{attribute 'global_init_slot' := '40510'}
VAR_GLOBAL
  LblAgg_FunctionallyIndependentEequipment                 :FB_BA_Label:=( sObjName:='FEE', sDescr:='Funktional eigenständige Einrichtung');
  LblAgg_SelfContainedControlUnit                          :FB_BA_Label:=( sObjName:='ASR', sDescr:='Autarke Steuer- oder Regeleinheit');
  LblAgg_ControlCabinet                                    :FB_BA_Label:=( sObjName:='SSK', sDescr:='Schaltschrank (gewerkespezifisch)');
//     330 Türen, Tore, Fenster, Sonnenschutz
  LblAgg_WindowDrive                                       :FB_BA_Label:=( sObjName:='FEN', sDescr:='Fenster (Antrieb)');
  LblAgg_WindowContact                                     :FB_BA_Label:=( sObjName:='FEK', sDescr:='Fensterkontakt');
  LblAgg_Blind                                             :FB_BA_Label:=( sObjName:='JAL', sDescr:='Jalousie');
  LblAgg_Awning                                            :FB_BA_Label:=( sObjName:='MAR', sDescr:='Markise');
  LblAgg_RollerShutters                                    :FB_BA_Label:=( sObjName:='ROL', sDescr:='Rollläden');
  LblAgg_Gate                                              :FB_BA_Label:=( sObjName:='TOR', sDescr:='Tor');
  LblAgg_Door                                              :FB_BA_Label:=( sObjName:='TÜR', sDescr:='Tür');
  LblAgg_DoorContact                                       :FB_BA_Label:=( sObjName:='TÜK', sDescr:='Türkontakt');
  LblAgg_Blackout                                          :FB_BA_Label:=( sObjName:='VER', sDescr:='Verdunklung');
//     412 Wasseranlagen
  LblAgg_TraceHeating                                      :FB_BA_Label:=( sObjName:='BGH', sDescr:='Begleitheizung');
  LblAgg_ElectricHeating                                   :FB_BA_Label:=( sObjName:='EWH', sDescr:='Elektroheizung (TWW–Bereitung)');
  LblAgg_WaterFilter                                       :FB_BA_Label:=( sObjName:='WFL', sDescr:='Wasserfilter');
//     421 Wärmeerzeugungsanlagen
  LblAgg_Furnace                                           :FB_BA_Label:=( sObjName:='HZK', sDescr:='Heizkessel');
  LblAgg_HeatExchanger                                     :FB_BA_Label:=( sObjName:='WÜT', sDescr:='Wärmeübertrager');
//     430 Lufttechnische Anlagen und Kälteanlagen
  LblAgg_FanExhaustAir                                     :FB_BA_Label:=( sObjName:='FOV', sDescr:='Fortluftventilator');
  LblAgg_Airwasher                                         :FB_BA_Label:=( sObjName:='LWS', sDescr:='Luftwäscher');
  LblAgg_Humidifier                                        :FB_BA_Label:=( sObjName:='BEF', sDescr:='Befeuchter');
  LblAgg_HumidifierPump                                    :FB_BA_Label:=( sObjName:='BFP', sDescr:='Befeuchterpumpe');
  LblAgg_FireDamper                                        :FB_BA_Label:=( sObjName:='BSK', sDescr:='Brandschutzklappe, -ventil');
  LblAgg_SmokeProtectionDamper                             :FB_BA_Label:=( sObjName:='RSK', sDescr:='Rauchschutzklappe');
  LblAgg_SmokeExtractorDamper                              :FB_BA_Label:=( sObjName:='ERK', sDescr:='Entrauchungsklappe');
  LblAgg_CeilingSwirlDiffuser                              :FB_BA_Label:=( sObjName:='DDA', sDescr:='Deckendrallauslass');
  LblAgg_RoofAirHeater                                     :FB_BA_Label:=( sObjName:='DLA', sDescr:='Deckenlufterhitzer');
  LblAgg_DirectEvaporator                                  :FB_BA_Label:=( sObjName:='DVD', sDescr:='Direktverdampfer');
  LblAgg_ElectricalAirHeater                               :FB_BA_Label:=( sObjName:='ELH', sDescr:='Elektrolufterhitzer');
  LblAgg_ElectricReHeater                                  :FB_BA_Label:=( sObjName:='ENH', sDescr:='Elektronacherhitzer');
  LblAgg_ElectricaPreHeater                                :FB_BA_Label:=( sObjName:='EVH', sDescr:='Elektrovorerhitzer');
  LblAgg_HeaterGeneral                                     :FB_BA_Label:=( sObjName:='ERH', sDescr:='Erhitzer');
  LblAgg_FanExtractAir                                     :FB_BA_Label:=( sObjName:='ABV', sDescr:='Abluftventilator');
  LblAgg_InductionDevice                                   :FB_BA_Label:=( sObjName:='IND', sDescr:='Induktionsgerät');
  LblAgg_RefrigerantDryer                                  :FB_BA_Label:=( sObjName:='KTR', sDescr:='Kältetrockner');
  LblAgg_CirculatorySystem                                 :FB_BA_Label:=( sObjName:='KVS', sDescr:='KVS (WRG über Kreislaufverbundsysteme)');
  LblAgg_AirFilterOutsideAir                               :FB_BA_Label:=( sObjName:='LFI', sDescr:='Außenluftfilter');
  LblAgg_AirFilterSupplyAir                                :FB_BA_Label:=( sObjName:='LFI', sDescr:='Zuluftfilter');
  LblAgg_AirFilterExhaustAir                               :FB_BA_Label:=( sObjName:='LFI', sDescr:='Fortluftfilter');
  LblAgg_AirFilterExtractAir                               :FB_BA_Label:=( sObjName:='LFI', sDescr:='Abluftfilter');
  LblAgg_AirFilter                                         :FB_BA_Label:=( sObjName:='LFI', sDescr:='Luftfilter');
  LblAgg_VentilationDamper                                 :FB_BA_Label:=( sObjName:='LKL', sDescr:='Lüftungsklappe');
  LblAgg_VentilationDamperOutsideAir                       :FB_BA_Label:=( sObjName:='LKL', sDescr:='Außenluftklappe');
  LblAgg_VentilationDamperExhaustAir                       :FB_BA_Label:=( sObjName:='LKL', sDescr:='Fortluftklappe');
  LblAgg_VentilationDamperMixAir                           :FB_BA_Label:=( sObjName:='LKL', sDescr:='Mischluftklappe');
  LblAgg_VentilationDamperSupplyAir                        :FB_BA_Label:=( sObjName:='LKL', sDescr:='Zuluftklappe');
  LblAgg_VentilationDamperBypassAir                        :FB_BA_Label:=( sObjName:='LKL', sDescr:='Bypassklappe');
  LblAgg_Pump                                              :FB_BA_Label:=( sObjName:='PPE', sDescr:='Pumpe');
  LblAgg_RecirculatingAirCoolingDevice                     :FB_BA_Label:=( sObjName:='ULK', sDescr:='Umluftkühlgerät');
  LblAgg_FanRecirculatingAir                               :FB_BA_Label:=( sObjName:='UMV', sDescr:='Umluftventilator');
  LblAgg_UvFilter                                          :FB_BA_Label:=( sObjName:='UVF', sDescr:='UV-Filter');
  LblAgg_VariableFlowRateController                        :FB_BA_Label:=( sObjName:='VVR', sDescr:='Variabler Volumenstromregler');
  LblAgg_WaterAirHeater                                    :FB_BA_Label:=( sObjName:='WLH', sDescr:='Wasserlufterhitzer');
  LblAgg_WaterReHeater                                     :FB_BA_Label:=( sObjName:='WNH', sDescr:='Wassernacherhitzer');
  LblAgg_WaterPreHeater                                    :FB_BA_Label:=( sObjName:='WVH', sDescr:='Wasservorerhitzer');
  LblAgg_HeatRecovery                                      :FB_BA_Label:=( sObjName:='WRG', sDescr:='Wärmerückgewinnung');
  LblAgg_FanSupplyAir                                      :FB_BA_Label:=( sObjName:='ZUV', sDescr:='Zuluftventilator');
  LblAgg_SmokeExtractionSystems                            :FB_BA_Label:=( sObjName:='ERA', sDescr:='Entrauchungsanlagen');
  LblAgg_SmokeExtractionVentilator                         :FB_BA_Label:=( sObjName:='ERV', sDescr:='Entrauchungsventilator');
  LblAgg_VentWindow                                        :FB_BA_Label:=( sObjName:='NSF', sDescr:='Nachströmfenster');
  LblAgg_VentFlap                                          :FB_BA_Label:=( sObjName:='NSK', sDescr:='Nachströmklappe');
  LblAgg_VentDoor                                          :FB_BA_Label:=( sObjName:='NST', sDescr:='Nachströmtür');
  LblAgg_WakeFan                                           :FB_BA_Label:=( sObjName:='NSV', sDescr:='Nachströmventilator');
//     434 Kälteanlagen
  LblAgg_GlycoOilProtector                                 :FB_BA_Label:=( sObjName:='GLP', sDescr:='Glykol/Ölprotektor');
  LblAgg_Chiller                                           :FB_BA_Label:=( sObjName:='KMA', sDescr:='Kältemaschine');
  LblAgg_ReCoolingPlant                                    :FB_BA_Label:=( sObjName:='RKW', sDescr:='Rückkühlwerk');
//     440 Starkstromanlagen
  LblAgg_GeneralPowerSupply                                :FB_BA_Label:=( sObjName:='ASV', sDescr:='Allgemeine Spannungsversorgung');
  LblAgg_CombindeHeatPowerStation                          :FB_BA_Label:=( sObjName:='BHK', sDescr:='Blockheizkraftwerk');
  LblAgg_CompensationSystem                                :FB_BA_Label:=( sObjName:='KOA', sDescr:='Kompensationsanlage');
  LblAgg_CouplingSwitch                                    :FB_BA_Label:=( sObjName:='KUS', sDescr:='Kuppelschalter');
  LblAgg_LoadBreakSwitch                                   :FB_BA_Label:=( sObjName:='LTS', sDescr:='Lasttrennschalter');
  LblAgg_CircuitBreaker                                    :FB_BA_Label:=( sObjName:='LSS', sDescr:='Leistungsschalter');
  LblAgg_NetworkAnalyser                                   :FB_BA_Label:=( sObjName:='NAG', sDescr:='Netzanalysegerät');
  LblAgg_EmergencyPoweGeneratorUnit                        :FB_BA_Label:=( sObjName:='NSG', sDescr:='Notstromaggregat');
  LblAgg_EmergencyLighting                                 :FB_BA_Label:=( sObjName:='SIB', sDescr:='Sicherheitsbeleuchtung');
  LblAgg_SafetyPowerSupply                                 :FB_BA_Label:=( sObjName:='SSV', sDescr:='Sicherheitsspannungsversorgung');
  LblAgg_Transformer                                       :FB_BA_Label:=( sObjName:='TRF', sDescr:='Transformator');
  LblAgg_UninterruptiblePowerSupply                        :FB_BA_Label:=( sObjName:='USV', sDescr:='Unterbrechungsfreie Spannungsversorgung');
//     450 Fernmelde- und informationstechnische Anlagen
  LblAgg_CentralFireAlarmSystem                            :FB_BA_Label:=( sObjName:='BMZ', sDescr:='Brandmeldezentrale');
  LblAgg_FireControlPanel                                  :FB_BA_Label:=( sObjName:='FWT', sDescr:='Feuerwehrtableau');
  LblAgg_KitchenTableau                                    :FB_BA_Label:=( sObjName:='KÜT', sDescr:='Küchentableau');
  LblAgg_SmokeDetector                                     :FB_BA_Label:=( sObjName:='RME', sDescr:='Rauchmelder');
  LblAgg_SmokeProtectionScreen                             :FB_BA_Label:=( sObjName:='RSV', sDescr:='Rauchschutzvorhang');
  LblAgg_VoiceAlarmCentre                                  :FB_BA_Label:=( sObjName:='SAZ', sDescr:='Sprachalarmierungszentrale');
  LblAgg_Tableau                                           :FB_BA_Label:=( sObjName:='TBL', sDescr:='Tableau (allgemein)');
//     460 Förderanlagen
  LblAgg_LiftGeneral                                       :FB_BA_Label:=( sObjName:='AZA', sDescr:='Aufzug allgemein');
  LblAgg_GoodsLift                                         :FB_BA_Label:=( sObjName:='AZL', sDescr:='Lastenaufzug');
  LblAgg_PassengerLift                                     :FB_BA_Label:=( sObjName:='AZP', sDescr:='Personenaufzug');
//     470 Nutzerspezifische Anlagen
  LblAgg_FumeCupboard                                      :FB_BA_Label:=( sObjName:='DIG', sDescr:='Digestorium');
  LblAgg_Compressor                                        :FB_BA_Label:=( sObjName:='KOM', sDescr:='Kompressor');
  LblAgg_ProgrammableLogicControllers                      :FB_BA_Label:=( sObjName:='SPS', sDescr:='Speicherprogrammierbare Steuerung');
//     479 Nutzerspezifische Anlage, Wetterstation
  LblAgg_RainSensor                                        :FB_BA_Label:=( sObjName:='RGM', sDescr:='Regenmelder');
  LblAgg_SolarRadiation                                    :FB_BA_Label:=( sObjName:='SES', sDescr:='Sonneneinstrahlung');
  LblAgg_WeatherStation                                    :FB_BA_Label:=( sObjName:='WST', sDescr:='Wetterstation');
  LblAgg_WindSpeed                                         :FB_BA_Label:=( sObjName:='WDG', sDescr:='Windgeschwindigkeit');
  LblAgg_WindDirection                                     :FB_BA_Label:=( sObjName:='WDR', sDescr:='Windrichtung');
  LblAgg_WindForce                                         :FB_BA_Label:=( sObjName:='WDS', sDescr:='Windstärke');
  LblAgg_Brightness                                        :FB_BA_Label:=( sObjName:='HEL', sDescr:='Helligkeit');
  LblAgg_Dawn                                              :FB_BA_Label:=( sObjName:='HED', sDescr:='Dämmerungshelligkeit');
  LblAgg_PressureAbsolute                                  :FB_BA_Label:=( sObjName:='LUA', sDescr:='Luftdruck absolut');
  LblAgg_PressureRelative                                  :FB_BA_Label:=( sObjName:='LUR', sDescr:='Luftdruck relativ');
  LblAgg_GeoLatitude                                       :FB_BA_Label:=( sObjName:='BRG', sDescr:='Breitengrad');
  LblAgg_GeoLongitude                                      :FB_BA_Label:=( sObjName:='LAG', sDescr:='Längengrad');
  LblAgg_SunAzimuth                                        :FB_BA_Label:=( sObjName:='SST', sDescr:='Sonnenstand');
  LblAgg_SunElevation                                      :FB_BA_Label:=( sObjName:='SEL', sDescr:='Elevation');
  LblAgg_WeatherStationReset                               :FB_BA_Label:=( sObjName:='ALS', sDescr:='Wetterstation Reset');
  LblAgg_WeatherStationCommReset                           :FB_BA_Label:=( sObjName:='ALS', sDescr:='Wetterstation Reset serielle Kommunikation');
  LblAgg_WeatherStationComm                                :FB_BA_Label:=( sObjName:='WST', sDescr:='Wetterstation Kommunikation');
//     480 Gebäudeautomation
  LblAgg_SystemSwitch                                      :FB_BA_Label:=( sObjName:='ANL', sDescr:='Anlagenschalter');
  LblAgg_AutomationStationEquipment                        :FB_BA_Label:=( sObjName:='ASE', sDescr:='Automationsstationseinrichtung');
  LblAgg_BusLineCoupler                                    :FB_BA_Label:=( sObjName:='BUS', sDescr:='Bus-Linien-Koppler');
  LblAgg_DataInterfaceUnit                                 :FB_BA_Label:=( sObjName:='DSE', sDescr:='Datenschnittstelleneinheit');
  LblAgg_FieldbusModule                                    :FB_BA_Label:=( sObjName:='FBM', sDescr:='Feldbusmodul');
  LblAgg_InformationFocalPoint                             :FB_BA_Label:=( sObjName:='ISP', sDescr:='Informationsschwerpunkt');
  LblAgg_ManagementAndControlEquipment                     :FB_BA_Label:=( sObjName:='MBE', sDescr:='Management- und Bedieneinrichtung');
//     481 GA-Sensorik – Temperatur
  LblAgg_TemperatureGasEmission                            :FB_BA_Label:=( sObjName:='TAG', sDescr:='Abgastemperatur');
  LblAgg_TemperatureExtractAir                             :FB_BA_Label:=( sObjName:='TAB', sDescr:='Ablufttemperatur');
  LblAgg_TemperatureOutside                                :FB_BA_Label:=( sObjName:='TAU', sDescr:='Außentemperatur');
  LblAgg_TemperatureExhaustAir                             :FB_BA_Label:=( sObjName:='TFO', sDescr:='Fortlufttemperatur');
  LblAgg_FrostProtectionMonitor                            :FB_BA_Label:=( sObjName:='FSW', sDescr:='Frostschutzwächter');
  LblAgg_TemperatureMixedAir                               :FB_BA_Label:=( sObjName:='TMI', sDescr:='Mischlufttemperatur');
  LblAgg_TemperatureRoomAir                                :FB_BA_Label:=( sObjName:='TRU', sDescr:='Raumtemperatur');
  LblAgg_TemperatureReturnFlow                             :FB_BA_Label:=( sObjName:='TRL', sDescr:='Rücklauftemperatur');
  LblAgg_LimiterSafetyTemperature                          :FB_BA_Label:=( sObjName:='STB', sDescr:='Sicherheitstemperaturbegrenzer');
  LblAgg_MonitorSafetyTemperature                          :FB_BA_Label:=( sObjName:='STW', sDescr:='Sicherheitstemperaturwächter');
  LblAgg_TemperatureStorage                                :FB_BA_Label:=( sObjName:='TSP', sDescr:='Speichertemperatur');
  LblAgg_TemperatureDewPoint                               :FB_BA_Label:=( sObjName:='TTP', sDescr:='Taupunkttemperatur');
  LblAgg_MonitorDewPoint                                   :FB_BA_Label:=( sObjName:='TPW', sDescr:='Taupunktwächter');
  LblAgg_TemperatureAfterCooler                            :FB_BA_Label:=( sObjName:='TNK', sDescr:='Temperatur nach Kühler');
  LblAgg_TemperatureAfterPreHeater                         :FB_BA_Label:=( sObjName:='TNV', sDescr:='Temperatur nach Vorerhitzer');
  LblAgg_TemperatureAfterHeatRecovery                      :FB_BA_Label:=( sObjName:='TNW', sDescr:='Temperatur nach Wärmerückgewinnung');
  LblAgg_Thermostat                                        :FB_BA_Label:=( sObjName:='THM', sDescr:='Thermostat');
  LblAgg_TemperatureHotWater                               :FB_BA_Label:=( sObjName:='TWW', sDescr:='Temperatur Warmwasser');
  LblAgg_TemperatureCirculation                            :FB_BA_Label:=( sObjName:='TWZ', sDescr:='Temperatur Zirkulation');
  LblAgg_TemperatureRecirculatingAir                       :FB_BA_Label:=( sObjName:='TUM', sDescr:='Umlufttemperatur');
  LblAgg_TemperatureFlow                                   :FB_BA_Label:=( sObjName:='TVL', sDescr:='Vorlauftemperatur');
  LblAgg_TemperatureSupplyAir                              :FB_BA_Label:=( sObjName:='TZU', sDescr:='Zulufttemperatur');
  LblAgg_TemperatureWetBulp                                :FB_BA_Label:=( sObjName:='TFK', sDescr:='Feuchtkugeltemperatur');
  LblAgg_TemperatureWetBulpExtractAir                      :FB_BA_Label:=( sObjName:='FAB', sDescr:='Feuchtkugeltemperatur Abluft');
  LblAgg_TemperatureWetBulpExhaustAir                      :FB_BA_Label:=( sObjName:='FFO', sDescr:='Feuchtkugeltemperatur Fortluft');
  LblAgg_TemperatureWetBulpOutsideAir                      :FB_BA_Label:=( sObjName:='FAU', sDescr:='Feuchtkugeltemperatur Aussenluft');
  LblAgg_TemperatureWetBulpRoomAir                         :FB_BA_Label:=( sObjName:='FRU', sDescr:='Feuchtkugeltemperatur Raumluft');
  LblAgg_TemperatureWetBulpSupplyAir                       :FB_BA_Label:=( sObjName:='FZU', sDescr:='Feuchtkugeltemperatur Zuluft');
  LblAgg_TemperatureDewPointExtractAir                     :FB_BA_Label:=( sObjName:='TPA', sDescr:='Taupunkttemperatur Abluft');
  LblAgg_TemperatureDewPointExhaustAir                     :FB_BA_Label:=( sObjName:='TPF', sDescr:='Taupunkttemperatur Fortluft');
  LblAgg_TemperatureDewPointOutsideAir                     :FB_BA_Label:=( sObjName:='TPW', sDescr:='Taupunkttemperatur Aussenluft');
  LblAgg_TemperatureDewPointRoomAir                        :FB_BA_Label:=( sObjName:='TPR', sDescr:='Taupunkttemperatur Raumluft');
  LblAgg_TemperatureDewPointSupplyAir                      :FB_BA_Label:=( sObjName:='TPZ', sDescr:='Taupunkttemperatur Zuluft');
//     481 GA-Sensorik – Druck
  LblAgg_PressureExtractAir                                :FB_BA_Label:=( sObjName:='PAB', sDescr:='Abluftdruck');
  LblAgg_PressureOutsideAir                                :FB_BA_Label:=( sObjName:='PAU', sDescr:='Außenluftdruck');
  LblAgg_PressureDifferential                              :FB_BA_Label:=( sObjName:='PDI', sDescr:='Differenzdruck');
  LblAgg_PressureDifferentialOutsideAirFilter              :FB_BA_Label:=( sObjName:='PDI', sDescr:='Differenzdruck Außenluftfilter');
  LblAgg_PressureDifferentialExtractAirFilter              :FB_BA_Label:=( sObjName:='PDI', sDescr:='Differenzdruck Abluftfilter');
  LblAgg_PressureDifferentialExhaustAirFilter              :FB_BA_Label:=( sObjName:='PDI', sDescr:='Differenzdruck Fortluftfilter');
  LblAgg_PressureDifferentialSupplyAirFan                  :FB_BA_Label:=( sObjName:='PDI', sDescr:='Differenzdruck Zuluftventilator');
  LblAgg_PressureDifferentialExtractAirFan                 :FB_BA_Label:=( sObjName:='PDI', sDescr:='Differenzdruck Abluftventilator');
  LblAgg_PressureDifferentialExhaustAirFan                 :FB_BA_Label:=( sObjName:='PDI', sDescr:='Differenzdruck Fortluftventilator');
  LblAgg_PressureSensorFlow                                :FB_BA_Label:=( sObjName:='PVL', sDescr:='Drucksensor (Wasser) Vorlauf');
  LblAgg_MonitorPressure                                   :FB_BA_Label:=( sObjName:='DRW', sDescr:='Druckwächter');
  LblAgg_PressureExhaustAir                                :FB_BA_Label:=( sObjName:='PFO', sDescr:='Fortluftdruck');
  LblAgg_PressureRoomAir                                   :FB_BA_Label:=( sObjName:='PRU', sDescr:='Raumdruck');
  LblAgg_PressureIndexCircuitSensorDifferential            :FB_BA_Label:=( sObjName:='PSI', sDescr:='Schlechtpunktfühler Differenzdruck');
  LblAgg_LimiterSafetyPressure                             :FB_BA_Label:=( sObjName:='SDB', sDescr:='Sicherheitsdruckbegrenzer');
  LblAgg_PressureSupplyAir                                 :FB_BA_Label:=( sObjName:='PZU', sDescr:='Zuluftdruck');
//     481 GA-Sensorik – Luftqualität
  LblAgg_CO2Sensor                                         :FB_BA_Label:=( sObjName:='COM', sDescr:='CO2-Sensor');
  LblAgg_CO2ExtractAir                                     :FB_BA_Label:=( sObjName:='CAB', sDescr:='CO2 Abluft');
  LblAgg_CO2ExhaustAir                                     :FB_BA_Label:=( sObjName:='CFO', sDescr:='CO2 Fortluft');
  LblAgg_CO2OutsideAir                                     :FB_BA_Label:=( sObjName:='CAU', sDescr:='CO2 Aussenluft');
  LblAgg_CO2RoomAir                                        :FB_BA_Label:=( sObjName:='CRU', sDescr:='CO2 Raum');
  LblAgg_CO2SupplyAir                                      :FB_BA_Label:=( sObjName:='CZU', sDescr:='CO2 Zuluft');
  LblAgg_QualityExtractAir                                 :FB_BA_Label:=( sObjName:='QAB', sDescr:='Luftqualität Abluft');
  LblAgg_QualityExhaustAir                                 :FB_BA_Label:=( sObjName:='QFO', sDescr:='Luftqualität Fortluft');
  LblAgg_QualityOutsideAir                                 :FB_BA_Label:=( sObjName:='QAU', sDescr:='Luftqualität Aussenluft');
  LblAgg_OualityRoomAir                                    :FB_BA_Label:=( sObjName:='QRU', sDescr:='Luftqualität Raum');
  LblAgg_QualitiySupplyAir                                 :FB_BA_Label:=( sObjName:='QZU', sDescr:='Luftqualität Zuluft');
  LblAgg_QualityAirSensor                                  :FB_BA_Label:=( sObjName:='LQF', sDescr:='Luftqualitätsfühler');
//     481 GA-Sensorik – Feuchte
  LblAgg_Hygrostat                                         :FB_BA_Label:=( sObjName:='HYG', sDescr:='Hygrostat');
  LblAgg_RelativeHumidityExtractAir                        :FB_BA_Label:=( sObjName:='MAB', sDescr:='Abluftfeuchte relativ');
  LblAgg_RelativeHumidityOutsideAir                        :FB_BA_Label:=( sObjName:='MAU', sDescr:='Außenfeuchte relativ');
  LblAgg_RelativeHumidityExhaustAir                        :FB_BA_Label:=( sObjName:='MFO', sDescr:='Fortluftfeuchte relativ');
  LblAgg_MonitorCondensation                               :FB_BA_Label:=( sObjName:='MKW', sDescr:='Kondensationswächter');
  LblAgg_RelativeHumidityMixedAir                          :FB_BA_Label:=( sObjName:='MMI', sDescr:='Mischluftfeuchte relativ');
  LblAgg_RelativeHumidityRoomHumidity                      :FB_BA_Label:=( sObjName:='MRU', sDescr:='Raumfeuchte relativ');
  LblAgg_RelativeHumidityRecirculatedAir                   :FB_BA_Label:=( sObjName:='MUM', sDescr:='Umluftfeuchte relativ');
  LblAgg_RelativeHumiditySupplyAir                         :FB_BA_Label:=( sObjName:='MZU', sDescr:='Zuluftfeuchte relativ');
  LblAgg_AbsoluteHumidityExtractAir                        :FB_BA_Label:=( sObjName:='XAB', sDescr:='Abluftfeuchte absolut');
  LblAgg_AbsoluteHumidityOutsideAir                        :FB_BA_Label:=( sObjName:='XAU', sDescr:='Außenluftfeuchte absolut');
  LblAgg_AbsoluteHumidityExhaustAir                        :FB_BA_Label:=( sObjName:='XFO', sDescr:='Fortluftfeuchte absolut');
  LblAgg_AbsoluteHumidityMixedAir                          :FB_BA_Label:=( sObjName:='XMI', sDescr:='Mischluftfeuchte absolut');
  LblAgg_AbsoluteHumidityRoomAir                           :FB_BA_Label:=( sObjName:='XRU', sDescr:='Raumfeuchte absolut');
  LblAgg_AbsoluteHumidityRecirculatingAir                  :FB_BA_Label:=( sObjName:='XUM', sDescr:='Umluftfeuchte absolut');
  LblAgg_AbsoluteHumiditySupplyAir                         :FB_BA_Label:=( sObjName:='XZU', sDescr:='Zuluftfeuchte absolut');
//     481 GA-Sensorik – Verbrauchserfassung
  LblAgg_MeterElectric                                     :FB_BA_Label:=( sObjName:='ELZ', sDescr:='Elektrozähler');
  LblAgg_MeterGasNaturalGas                                :FB_BA_Label:=( sObjName:='EGZ', sDescr:='Gaszähler Erdgas');
  LblAgg_MeterCoolingEnergy                                :FB_BA_Label:=( sObjName:='KMZ', sDescr:='Kältemengenzähler');
  LblAgg_MeterHeat                                         :FB_BA_Label:=( sObjName:='WMZ', sDescr:='Wärmemengenzähler');
  LblAgg_MetferWater                                       :FB_BA_Label:=( sObjName:='WAZ', sDescr:='Wasserzähler');
  LblAgg_MeterFuel                                         :FB_BA_Label:=( sObjName:='BSZ', sDescr:='Brennstoffzähler (Öl)');
  LblAgg_MeterSteam                                        :FB_BA_Label:=( sObjName:='DMZ', sDescr:='Dampfmengenzähler');
  LblAgg_DegreeDayNumber                                   :FB_BA_Label:=( sObjName:='GTZ', sDescr:='Gradtagszahl');
//     481 GA-Sensorik – Zustandserfassung und sonstige
  LblAgg_LeakageMonitoring                                 :FB_BA_Label:=( sObjName:='LCK', sDescr:='Leckageüberwachung');
  LblAgg_EmergencyStop                                     :FB_BA_Label:=( sObjName:='NOT', sDescr:='Not-Aus-Einrichtung/-Taster');
  LblAgg_StockLevel                                        :FB_BA_Label:=( sObjName:='LSP', sDescr:='Speicherfüllstand');
  LblAgg_FlowMonitor                                       :FB_BA_Label:=( sObjName:='SSW', sDescr:='Strömungswächter');
  LblAgg_OverflowMonitoring                                :FB_BA_Label:=( sObjName:='UBL', sDescr:='Überlaufüberwachung');
  LblAgg_LowWaterCutOff                                    :FB_BA_Label:=( sObjName:='WMS', sDescr:='Wassermangelsicherung');
  LblAgg_WaterFlowMonitor                                  :FB_BA_Label:=( sObjName:='WSW', sDescr:='Wasserströmungswächter');
//     481 GA-Sensorik – Drehzahl
  LblAgg_PumpSpeed                                         :FB_BA_Label:=( sObjName:='SPP', sDescr:='Drehzahl Pumpe');
  LblAgg_FanSpeedExtractAir                                :FB_BA_Label:=( sObjName:='SAB', sDescr:='Drehzahl Ventilator (Abluft)');
  LblAgg_FanSpeedExhaustAir                                :FB_BA_Label:=( sObjName:='SFO', sDescr:='Drehzahl Ventilator (Fortluft)');
  LblAgg_FanSpeedSupplyAir                                 :FB_BA_Label:=( sObjName:='SZU', sDescr:='Drehzahl Ventilator (Zuluft)');
//     481 GA-Sensorik – Volumenstrom
  LblAgg_VolumeFlowRateExtractAir                          :FB_BA_Label:=( sObjName:='VAB', sDescr:='Volumenstrom Abluft');
  LblAgg_VolumeFlowRateOutsideAir                          :FB_BA_Label:=( sObjName:='VAU', sDescr:='Volumenstrom Außenluft');
  LblAgg_VolumeFlowRateExhaustAir                          :FB_BA_Label:=( sObjName:='VFO', sDescr:='Volumenstrom Fortluft');
  LblAgg_VolumeFlowRateBrineCirculatorySystem              :FB_BA_Label:=( sObjName:='VSO', sDescr:='Volumenstrom Sole (KVS)');
  LblAgg_VolumeFlowRateColdDrinkingWater                   :FB_BA_Label:=( sObjName:='VKW', sDescr:='Volumenstrom Trinkwasser kalt');
  LblAgg_VolumeFlowRateHotDrinkingWater                    :FB_BA_Label:=( sObjName:='VWW', sDescr:='Volumenstrom Trinkwasser warm');
  LblAgg_VolumeFlowRateWaterPurification                   :FB_BA_Label:=( sObjName:='VAW', sDescr:='Volumenstrom Wasseraufbereitung');
  LblAgg_VolumeFlowRateSupplyAir                           :FB_BA_Label:=( sObjName:='VZU', sDescr:='Volumenstrom Zuluft');
//     481 GA-Sensorik – Enthalpie
  LblAgg_Enthalpy                                          :FB_BA_Label:=( sObjName:='ETH', sDescr:='Enthalpie');
  LblAgg_EnthalpyExtractAir                                :FB_BA_Label:=( sObjName:='EAB', sDescr:='Enthalpie Abluft');
  LblAgg_EnthalpyExhaustAir                                :FB_BA_Label:=( sObjName:='EFO', sDescr:='Enthalpie Fortluft');
  LblAgg_EnthalpyOutsideAir                                :FB_BA_Label:=( sObjName:='EAU', sDescr:='Enthalpie Aussenluft');
  LblAgg_EnthalpyRoomAir                                   :FB_BA_Label:=( sObjName:='ERU', sDescr:='Enthalpie Raumluft');
  LblAgg_EnthalpySupplyAir                                 :FB_BA_Label:=( sObjName:='EZU', sDescr:='Enthalpie Zuluft');
//     481 GA-Sensorik – Multifunktionssensor
  LblAgg_MultiSensorExtractAir                             :FB_BA_Label:=( sObjName:='MAB', sDescr:='Multifunktionssensor Abluft');
  LblAgg_MultiSensorExhaustAir                             :FB_BA_Label:=( sObjName:='MFO', sDescr:='Multifunktionssensor Fortluft');
  LblAgg_MultiSensorOutsideAir                             :FB_BA_Label:=( sObjName:='MAU', sDescr:='Multifunktionssensor Aussenluft');
  LblAgg_MultiSensorRoomAir                                :FB_BA_Label:=( sObjName:='MRU', sDescr:='Multifunktionssensor Raum');
  LblAgg_MultiSensorSupplyAir                              :FB_BA_Label:=( sObjName:='MZU', sDescr:='Multifunktionssensor Zuluft');
//     481 GA-Aktorik – Stellantriebe
  LblAgg_ValveRadiator                                     :FB_BA_Label:=( sObjName:='HKV', sDescr:='Heizkörperventil-Antrieb');
  LblAgg_ValveCoolingCeiling                               :FB_BA_Label:=( sObjName:='KDV', sDescr:='Kühldeckenventil-Antrieb');
  LblAgg_MotorisedFlap                                     :FB_BA_Label:=( sObjName:='KLA', sDescr:='Motorische Klappe');
  LblAgg_Valve                                             :FB_BA_Label:=( sObjName:='VEN', sDescr:='Motorventil ');
  LblAgg_HumidifierValve                                   :FB_BA_Label:=( sObjName:='VEN', sDescr:='Befeuchter Ventil ');
//     481 GA-Beleuchtung
  LblAgg_IlluminationExternal                              :FB_BA_Label:=( sObjName:='EAU', sDescr:='Beleuchtungsstärke Außen');
  LblAgg_IlluminationRoom                                  :FB_BA_Label:=( sObjName:='ERU', sDescr:='Beleuchtungsstärke Raum');
  LblAgg_LightColourRoom                                   :FB_BA_Label:=( sObjName:='CRU', sDescr:='Lichtfarbe Raum');
  LblAgg_RedLightIntensity                                 :FB_BA_Label:=( sObjName:='LRT', sDescr:='Lichtintensität rot');
  LblAgg_GreenLightIntensity                               :FB_BA_Label:=( sObjName:='LGN', sDescr:='Lichtintensität grün');
  LblAgg_BlueLightIntensity                                :FB_BA_Label:=( sObjName:='LBL', sDescr:='Lichtintensität blau');
//     481 GA-Sonnenschutz
  LblAgg_BlindAnglePosition                                :FB_BA_Label:=( sObjName:='JWI', sDescr:='Winkelposition Jalousie');
  LblAgg_ShadingPosition                                   :FB_BA_Label:=( sObjName:='JPO', sDescr:='Verschattungsposition');
  LblAgg_MovementCommand                                   :FB_BA_Label:=( sObjName:='JFB', sDescr:='Jalousie Fahrbefehl');
//     485 Raumautomation
  LblAgg_DisplayAndControlUnit                             :FB_BA_Label:=( sObjName:='ABE', sDescr:='Anzeige- und Bedieneinrichtung');
  LblAgg_PresenceSwitches                                  :FB_BA_Label:=( sObjName:='PME', sDescr:='Präsenzschalter, -melder, Bewegungsmelder');
  LblAgg_RoomAutomationDevice                              :FB_BA_Label:=( sObjName:='RAE', sDescr:='Raumautomationseinrichtung');
  LblAgg_RoomControlUnit                                   :FB_BA_Label:=( sObjName:='RBG', sDescr:='Raumbediengerät');
//     Beckhoff ADS Kommunikation
  LblAgg_GeneralSettingsCom                                :FB_BA_Label:=( sObjName:='COM', sDescr:='Anlagenparameter Kommunikation');
  LblAgg_GeneralSettingsComDst                             :FB_BA_Label:=( sObjName:='WEK', sDescr:='Störung Allgemeine Daten');
  LblAgg_DataCommunicationExternalControl                  :FB_BA_Label:=( sObjName:='COM', sDescr:='Datenkommunikation Fremdsteuerung');
END_VAR

// ---- Templates/GVLs/Language/German/LblControl_DE.TcGVL
{region '#Template'}
	{attribute 'Version' := '5.0.0.0'}
	{attribute 'Tags' := '"LCID": "1031", "Text": "GVL, AKS, Labels, ObjectName, Description"'}
	{attribute 'Tags' := '"LCID": "1033", "Text": "GVL, DPAD, Labels, ObjectName, Description"'}
	{attribute 'Description' := '"LCID": "1031", "Text": "Anlagenkennzeichnungssystem, Labels controls"'}
	{attribute 'Description' := '"LCID": "1033", "Text": "Data Point Addressing Description, Labels controls"'}
{endregion}

{attribute 'global_init_slot' := '40510'}
VAR_GLOBAL
  LblCtl_OperationMode                                     :FB_BA_Label:=( sObjName:='BTA', sDescr:='Betriebsart');
  LblCtl_SummerNightCooling                                :FB_BA_Label:=( sObjName:='SNK', sDescr:='Sommernachtkühlung');
  LblCtl_DifferencePressureMonitoringSupplyAirFan          :FB_BA_Label:=( sObjName:='DRW', sDescr:='Zuluftventilator Differenzdrucküberwachung ');
  LblCtl_DifferencePressureMonitoringExtractAirFan         :FB_BA_Label:=( sObjName:='DRW', sDescr:='Abluftventilator Differenzdrucküberwachung ');
  LblCtl_TSetpointCalculation                              :FB_BA_Label:=( sObjName:='SWC', sDescr:='Sollwertberechnung Temperatur');
  LblCtl_HSetpointCalculation                              :FB_BA_Label:=( sObjName:='SWC', sDescr:='Sollwertberechnung Feuchte');
  LblCtl_TCascadeSupplyAirControl                          :FB_BA_Label:=( sObjName:='RGL', sDescr:='Führungsregelung Zulufttemperatur');
  LblCtl_HCascadeSupplyAirControl                          :FB_BA_Label:=( sObjName:='RGL', sDescr:='Führungsregelung Zuluftfeuchte');
  LblCtl_PreHeater                                         :FB_BA_Label:=( sObjName:='VEH', sDescr:='Vorerhitzer');
  LblCtl_ReHeater                                          :FB_BA_Label:=( sObjName:='NEH', sDescr:='Nacherhitzer');
  LblCtl_EnergyRecovery                                    :FB_BA_Label:=( sObjName:='ERG', sDescr:='Energierückgewinnung');
  LblCtl_SupplyAirTemperatureControl                       :FB_BA_Label:=( sObjName:='RGL', sDescr:='Zulufttemperaturregelung');
  LblCtl_SupplyAirDehumidifierControl                      :FB_BA_Label:=( sObjName:='RGL', sDescr:='Zuluftentfeuchtereglung');
  LblCtl_SupplyAirHumidifierController                     :FB_BA_Label:=( sObjName:='RGL', sDescr:='Zuluftfeuchtereglung');
  LblCtl_SupplyAirTemperatureLimitationControl             :FB_BA_Label:=( sObjName:='RGL', sDescr:='Zulufttemperatur Begrenzungsregelung ');
  LblCtl_ReturnWaterControl                                :FB_BA_Label:=( sObjName:='RGL', sDescr:='Rücklauftemperaturregelung');
  LblCtl_HumidityLimitationControl                         :FB_BA_Label:=( sObjName:='RGL', sDescr:='Rel Feuchte Begrenzungsregelung');
  LblCtl_CalculationPreRinseSetpoint                       :FB_BA_Label:=( sObjName:='SWB', sDescr:='Berechung Vorspülsollwert ');
  LblCtl_FrostProtectionControl                            :FB_BA_Label:=( sObjName:='FSR', sDescr:='Frostschutzregelung luftseitig');
  LblCtl_ExhaustAirTemperatureControl                      :FB_BA_Label:=( sObjName:='RGL', sDescr:='Fortlufttemperaturregelung');
  LblCtl_EnergyRecoveryDeicingRamp                         :FB_BA_Label:=( sObjName:='RMP', sDescr:='Rampe Enteisung');
  LblCtl_BACnetDevice                                      :FB_BA_Label:=( sObjName:='DEV', sDescr:='BACnet device');
  LblCtl_PlantControl                                      :FB_BA_Label:=( sObjName:='ALS', sDescr:='Anlagensteuerung');
  LblCtl_TSequenceControl                                  :FB_BA_Label:=( sObjName:='SEQ', sDescr:='Sequenzsteuerung Temp');
  LblCtl_HSequenceControl                                  :FB_BA_Label:=( sObjName:='SEQ', sDescr:='Sequenzsteuerung Feuchte');
  LblCtl_GeneralBeckhoffEventClass                         :FB_BA_Label:=( sObjName:='EKL', sDescr:='Ereignisklasse');
  LblCtl_GeneralSettings                                   :FB_BA_Label:=( sObjName:='ALP', sDescr:='Anlagenparameter');
  LblCtl_GeneralCabinetBasicEquipment                      :FB_BA_Label:=( sObjName:='SSG', sDescr:='Schaltschrank Grundausstattung');
  LblCtl_GeneralCabinetAdditionalEquipment                 :FB_BA_Label:=( sObjName:='SSZ', sDescr:='Schaltschrank Zusatzausstattung');
  LblCtl_EventIndicationLamp                               :FB_BA_Label:=( sObjName:='SMM', sDescr:='Sammelstörmeldung Lampe');
  LblCtl_AcknowledgeCommand                                :FB_BA_Label:=( sObjName:='QUI', sDescr:='Hardware quittieren');
  LblCtl_RemoteAcknowledgement                             :FB_BA_Label:=( sObjName:='QUI', sDescr:='Fernquittierung Störung');
  LblCtl_LocalAcknowledgement                              :FB_BA_Label:=( sObjName:='QUI', sDescr:='Lokale Quittierung Störung');
  LblCtl_Acknowledge                                       :FB_BA_Label:=( sObjName:='QUI', sDescr:='Quittierung');
//     
  LblCtl_Fuse                                              :FB_BA_Label:=( sObjName:='SIC', sDescr:='Sicherung');
//     Einstellungen
  LblCtl_FrostProtection                                   :FB_BA_Label:=( sObjName:='FRS', sDescr:='Frostschutz');
  LblCtl_MinimumOutsideTemperature                         :FB_BA_Label:=( sObjName:='TWI', sDescr:='Minimale Außentemperatur');
  LblCtl_TemperatureWeatherLowLimit                        :FB_BA_Label:=( sObjName:='TWI', sDescr:='Minimale Außentemperatur unterer Grenzwert');
  LblCtl_TemperatureWeatherDamped                          :FB_BA_Label:=( sObjName:='TWG', sDescr:='Temperatur Witterung gedämpft');
  LblCtl_TemperatureWeatherDampedLowLimit                  :FB_BA_Label:=( sObjName:='TWG', sDescr:='Temperatur Witterung gedämpft unterer Grenzwert');
  LblCtl_PressureControl                                   :FB_BA_Label:=( sObjName:='RGL', sDescr:='Druckregelung');
  LblCtl_Converter3Point                                   :FB_BA_Label:=( sObjName:='WDL', sDescr:='3 Punkt Wandler');
  LblCtl_HeatingCurve                                      :FB_BA_Label:=( sObjName:='HKV', sDescr:='Heizkurve');
  LblCtl_SetpointGeneration                                :FB_BA_Label:=( sObjName:='SWG', sDescr:='Sollwert Generierung');
  LblCtl_RequestHeatState                                  :FB_BA_Label:=( sObjName:='AWZ', sDescr:='Wärmeanforderung Zustand');
  LblCtl_RequestHeatSetpoint                               :FB_BA_Label:=( sObjName:='AWS', sDescr:='Wärmeanforderung Sollwert');
  LblCtl_FlowTempControl                                   :FB_BA_Label:=( sObjName:='RGL', sDescr:='Vorlauf Temperatur Regelung');
//     
  LblCtl_RoomTemperatureControl                            :FB_BA_Label:=( sObjName:='RGL', sDescr:='Raumtemperaturregelung');
  LblCtl_FlowTemperatureControl                            :FB_BA_Label:=( sObjName:='RGL', sDescr:='Vorlauftemperatur Regelung');
  LblCtl_HeatValve                                         :FB_BA_Label:=( sObjName:='VEN', sDescr:='Ventil heizen');
  LblCtl_CoolValve                                         :FB_BA_Label:=( sObjName:='VEN', sDescr:='Ventil kühlen');
  LblCtl_HeatingController                                 :FB_BA_Label:=( sObjName:='LPH', sDescr:='Heizregler');
  LblCtl_CoolingController                                 :FB_BA_Label:=( sObjName:='LPC', sDescr:='Kühlregler');
  LblCtl_Light                                             :FB_BA_Label:=( sObjName:='LIT', sDescr:='Licht');
  LblCtl_SetpointHeating                                   :FB_BA_Label:=( sObjName:='SWG', sDescr:='Sollwertgenerierung heizen');
  LblCtl_SetpointCooling                                   :FB_BA_Label:=( sObjName:='SWG', sDescr:='Sollwertgenerierung kühlen');
  LblCtl_Facade                                            :FB_BA_Label:=( sObjName:='FEE', sDescr:='Fassadendaten');
  LblCtl_BuildingAlarms                                    :FB_BA_Label:=( sObjName:='FEE', sDescr:='Gebäude Alarme');
  LblCtl_BuildingEnergyLevel                               :FB_BA_Label:=( sObjName:='FEE', sDescr:='Gebäude Energieniveaus');
  LblCtl_BuildingMode                                      :FB_BA_Label:=( sObjName:='FEE', sDescr:='Gebäude Betriebsmodus');
  LblCtl_BuildingSpRmT                                     :FB_BA_Label:=( sObjName:='FEE', sDescr:='Gebäude Raumtemperatursollwerte');
  LblCtl_BuildingSunprotection                             :FB_BA_Label:=( sObjName:='FEE', sDescr:='Gebäude Sonnenschutz');
  LblCtl_TemperatureFrost                                  :FB_BA_Label:=( sObjName:='TFR', sDescr:='Temperatur Frost');
  LblCtl_MixedAirStartUpRamp                               :FB_BA_Label:=( sObjName:='RMP', sDescr:='Rampe Anlagenstart');
  LblCtl_Cooler                                            :FB_BA_Label:=( sObjName:='KUE', sDescr:='Kühler');
  LblCtl_EvtCategoryLifeSafty                              :FB_BA_Label:=( sObjName:='EGF', sDescr:='Gefahr für Leben');
  LblCtl_EvtCategorySaftyMessage                           :FB_BA_Label:=( sObjName:='ESM', sDescr:='Sicherheitsmeldung');
  LblCtl_EvtCategoryAlarmMessage                           :FB_BA_Label:=( sObjName:='EAM', sDescr:='Alarmeldung');
  LblCtl_EvtCategoryFaultMessage                           :FB_BA_Label:=( sObjName:='EST', sDescr:='Störungsmeldung');
  LblCtl_EvtCategoryMaintenanceMessage                     :FB_BA_Label:=( sObjName:='EWA', sDescr:='Wartungsmeldung ');
  LblCtl_EvtCategorySystem                                 :FB_BA_Label:=( sObjName:='ESY', sDescr:='Systemmeldung');
  LblCtl_EvtCategoryManualOperation                        :FB_BA_Label:=( sObjName:='EHA', sDescr:='Handeingriff');
  LblCtl_EvtCategoryOther                                  :FB_BA_Label:=( sObjName:='ESO', sDescr:='Sonstige Meldungen');
  LblCtl_TrendLogging                                      :FB_BA_Label:=( sObjName:='TRA', sDescr:='Trend');
  LblCtl_WeatherParameters                                 :FB_BA_Label:=( sObjName:='PWI', sDescr:='Witterung Parameter');
  LblCtl_SetpointFrostProtection                           :FB_BA_Label:=( sObjName:='SW_', sDescr:='Sollwert Frostschutz');
  LblCtl_SetpointWeatherIcing                              :FB_BA_Label:=( sObjName:='SW_', sDescr:='Sollwert Vereisung');
  LblCtl_SetpointMinimumOutsideTemperature                 :FB_BA_Label:=( sObjName:='SWI', sDescr:='Sollwert Minimale Außentemperatur');
  LblCtl_MeanDamped                                        :FB_BA_Label:=( sObjName:='MWT', sDescr:='Mittelwert Außentemperatur gedämpft');
  LblCtl_OperationalMessageTemperatureWeatherLowLimit      :FB_BA_Label:=( sObjName:='BM_', sDescr:='Betriebsmeldung Außentemperatur unterer Grenzwert');
  LblCtl_OperationalMessageTemperatureWeatherDampedLowLimit:FB_BA_Label:=( sObjName:='BM_', sDescr:='Betriebsmeldung Außentemperatur gedämpft unterer Grenzwert');
  LblCtl_PlantStartup                                      :FB_BA_Label:=( sObjName:='AST', sDescr:='Anlagenstart');
  LblCtl_TimeDelayDampersClose                             :FB_BA_Label:=( sObjName:='ZV_', sDescr:='Zeitverzögerung Klappen schliessen, Auslaufen der Ventilatoren');
  LblCtl_TimeDelaySupplyAirFanOn                           :FB_BA_Label:=( sObjName:='ZV_', sDescr:='Zeitverzögerung Zuluftventilator Ein');
  LblCtl_TimeDelayExtractAirFanOn                          :FB_BA_Label:=( sObjName:='ZV_', sDescr:='Zeitverzögerung Abluftventilator Ein');
  LblCtl_TimeDelayTemperatureSequenceControlOn             :FB_BA_Label:=( sObjName:='ZV_', sDescr:='Zeitverzögerung Temperatur Sequenz Steuerung Ein');
  LblCtl_TimeDelayTemperatureSequenceControlOff            :FB_BA_Label:=( sObjName:='ZV_', sDescr:='Zeitverzögerung Temperatur Sequenz Steuerung Aus');
  LblCtl_TimeDelayHumiditySequenceControlOn                :FB_BA_Label:=( sObjName:='ZV_', sDescr:='Zeitverzögerung Feuchte Sequenz Steuerung Ein');
  LblCtl_TimeDelayEnableMonitoringLimitValues              :FB_BA_Label:=( sObjName:='ZV_', sDescr:='Zeitverzögerung Freigabe Überwachung Grenzwerte');
  LblCtl_StagesOfThePlantStartup                           :FB_BA_Label:=( sObjName:='STA', sDescr:='Stufen des Anlagenstarts');
//     Beckhoff Schaltschrank Grundausstattung
  LblCtl_SwitchingCommandCollectiveFaultSignalLamp         :FB_BA_Label:=( sObjName:='SB_', sDescr:='Sammelstörmeldung Lampe Schaltbefehl');
  LblCtl_SwitchingCommandHardwareAcknowledgement           :FB_BA_Label:=( sObjName:='SB_', sDescr:='Hardware quittieren Schaltbefehl');
  LblCtl_ButtonRemoteAcknowledgement                       :FB_BA_Label:=( sObjName:='TS_', sDescr:='Eingabe Fernquittierung');
  LblCtl_ButtonLocalAcknowledgement                        :FB_BA_Label:=( sObjName:='TS_', sDescr:='Taster Quittierung');
//     Beckhoff Heizkreis
  LblCtl_HeatingLimit                                      :FB_BA_Label:=( sObjName:='HGW', sDescr:='Heizgrenzwert');
  LblCtl_PresentOperationMode                              :FB_BA_Label:=( sObjName:='ABA', sDescr:='aktuelle Betriebsart');
  LblCtl_OperationModeSelection                            :FB_BA_Label:=( sObjName:='BAA', sDescr:='Betriebsartenauswahl');
//     Beckhoff Sommernachtkühlung
  LblCtl_HysteresisRoomTemperature                         :FB_BA_Label:=( sObjName:='HYS', sDescr:='Hysterese Raumtemperatur');
  LblCtl_OutsideTemperatureLowLimit                        :FB_BA_Label:=( sObjName:='MIN', sDescr:='minimale Außentemperatur');
  LblCtl_OffValueDifferenceOutsideInsightTemperature       :FB_BA_Label:=( sObjName:='MIN', sDescr:='Ausschaltwert von Differenz Außentemperatur - Raumtemperatur');
  LblCtl_OnValueDifferenceOutsideInsightTemperature        :FB_BA_Label:=( sObjName:='MAX', sDescr:='Einschaltwert von Differenz Außentemperatur - Raumtemperatur');
//     Beckhoff Klappen
  LblCtl_DriveTimeOpen                                     :FB_BA_Label:=( sObjName:='LZA', sDescr:='Laufzeit Auf');
  LblCtl_DriveTimeClose                                    :FB_BA_Label:=( sObjName:='LZZ', sDescr:='Laufzeit Zu ');
  LblCtl_DisturbanceFeedbackOpen                           :FB_BA_Label:=( sObjName:='SMA', sDescr:='Störung Rückmeldung Auf');
  LblCtl_DisturbanceFeedbackClose                          :FB_BA_Label:=( sObjName:='SMZ', sDescr:='Störung Rückmeldung Zu');
//     Beckhoff Differenzdrucküberwachung
  LblCtl_TimeDelay                                         :FB_BA_Label:=( sObjName:='ZV_', sDescr:='Verzögerung ');
  LblCtl_TimeDelayFeedback                                 :FB_BA_Label:=( sObjName:='ZVR', sDescr:='Verzögerung Rückmeldung');
  LblCtl_TimeDelayInterruptionFeedback                     :FB_BA_Label:=( sObjName:='ANV', sDescr:='Ansprechverzögerung ');
//     Beckhoff Vorspülen
  LblCtl_PreRinseDuration                                  :FB_BA_Label:=( sObjName:='VSP', sDescr:='Vorspüldauer');
  LblCtl_DisturbancePreRinse                               :FB_BA_Label:=( sObjName:='SM_', sDescr:='Meldung Störung Vorspülen');
  LblCtl_SetpointMinimalReturnWaterTemperature             :FB_BA_Label:=( sObjName:='SW_', sDescr:='Sollwert minimale Rücklauftemperatur');
//     Beckhoff  Rampe
  LblCtl_RampTimeUp                                        :FB_BA_Label:=( sObjName:='RPA', sDescr:='Rampenzeit auf');
  LblCtl_RampTimeDown                                      :FB_BA_Label:=( sObjName:='RPZ', sDescr:='Rampenzeit ab');
  LblCtl_CommandOpen                                       :FB_BA_Label:=( sObjName:='SB_', sDescr:='Schaltbefehl Auf');
  LblCtl_CommandClose                                      :FB_BA_Label:=( sObjName:='SB_', sDescr:='Schaltbefehl Zu');
  LblCtl_CalculatedValue                                   :FB_BA_Label:=( sObjName:='ERW', sDescr:='errechneter Wert');
  LblCtl_Value                                             :FB_BA_Label:=( sObjName:='WET', sDescr:='Wert');
//     Beckhoff Ereignisklassen
  LblCtl_EvtClass                                          :FB_BA_Label:=( sObjName:='MDK', sDescr:='Meldungsklasse');
  LblCtl_FlowSwitch                                        :FB_BA_Label:=( sObjName:='BM_', sDescr:='Betriebsmeldung Strömungswächter');
  LblCtl_SmokeAlarm                                        :FB_BA_Label:=( sObjName:='SM_', sDescr:='Störung Rauchalarm');
  LblCtl_SystemFailure                                     :FB_BA_Label:=( sObjName:='SM_', sDescr:='Störung Systemfehler');
  LblCtl_Contamination                                     :FB_BA_Label:=( sObjName:='SM_', sDescr:='Störung Kontamination');
  LblCtl_SwitchingCommandSmokeDetector                     :FB_BA_Label:=( sObjName:='SB_', sDescr:='Schaltbefehl Quittierung');
  LblCtl_ButtonReset                                       :FB_BA_Label:=( sObjName:='TS_', sDescr:='Taster Quittierung');
  LblCtl_OffsetNightSetpoint                               :FB_BA_Label:=( sObjName:='SNK', sDescr:='Offset Nachtabsenkung');
//     
  LblCtl_SetpointRelHumidityHumidification                 :FB_BA_Label:=( sObjName:='SW_', sDescr:='Sollwert Relative Feuchte Befeuchten');
  LblCtl_SetpointRelHumidityDehumidification               :FB_BA_Label:=( sObjName:='SW_', sDescr:='Sollwert Relative Feuchte Entfeuchten');
  LblCtl_SetpointAbsHumidityHumidification                 :FB_BA_Label:=( sObjName:='SWC', sDescr:='Sollwert Absolute Feuchte Befeuchten');
  LblCtl_SetpointAbsHumidityDehumidification               :FB_BA_Label:=( sObjName:='SWC', sDescr:='Sollwert Absolute Feuchte Entfeuchten');
  LblCtl_SetpointRelHumidity                               :FB_BA_Label:=( sObjName:='SW_', sDescr:='Sollwert Relative Feuchte');
  LblCtl_SetpointAbsHumidity                               :FB_BA_Label:=( sObjName:='SW_', sDescr:='Sollwert Absolute Feuchte');
  LblCtl_OperationalMessageDehumidification                :FB_BA_Label:=( sObjName:='BM_', sDescr:='Betriebsmeldung Entfeuchtung');
//     
  LblCtl_SetpointSunblindPosition                          :FB_BA_Label:=( sObjName:='SW_', sDescr:='Sollwert Jalousie Position');
  LblCtl_SetpointSunblindAngle                             :FB_BA_Label:=( sObjName:='SW_', sDescr:='Sollwert Jalousie Winkel');
  LblCtl_CommandSunblindStart                              :FB_BA_Label:=( sObjName:='SB_', sDescr:='Startbefehl');
  LblCtl_ButtonSunblind                                    :FB_BA_Label:=( sObjName:='TS_', sDescr:='Jalousietaster');
  LblCtl_FeedbackSunblindPosition                          :FB_BA_Label:=( sObjName:='RM_', sDescr:='Rückmeldung Jalousie Position');
  LblCtl_FeedbackSunblindAngle                             :FB_BA_Label:=( sObjName:='RM_', sDescr:='Rückmeldung Jalousie Winkel');
  LblCtl_FeedbackSunblindPrio                              :FB_BA_Label:=( sObjName:='RM_', sDescr:='Rückmeldung Telegrammpriorität');
//     
  LblCtl_TimeDelayStormOn                                  :FB_BA_Label:=( sObjName:='ESV', sDescr:='Sturmerkennung Verzögerung Ein');
  LblCtl_TimeDelayStormOff                                 :FB_BA_Label:=( sObjName:='ASV', sDescr:='Sturmerkennung Verzögerung Aus');
  LblCtl_MaintenanceEnable                                 :FB_BA_Label:=( sObjName:='FRG', sDescr:='Wartungsposition Freigabe');
  LblCtl_MaintenancePosition                               :FB_BA_Label:=( sObjName:='SW_', sDescr:='Sollwert Wartung Position');
  LblCtl_MaintenanceAngle                                  :FB_BA_Label:=( sObjName:='SW_', sDescr:='Sollwert Wartung Winkel');
  LblCtl_FacadeThermoAutomaticEnable                       :FB_BA_Label:=( sObjName:='FRG', sDescr:='Fassaden-Thermoautomatik Freigabe');
  LblCtl_FacadeThermoAutomaticCoolingPosition              :FB_BA_Label:=( sObjName:='SW_', sDescr:='Fassaden-Thermoautomatik Kühl-Position');
  LblCtl_FacadeThermoAutomaticCoolingAngle                 :FB_BA_Label:=( sObjName:='SW_', sDescr:='Fassaden-Thermoautomatik Kühl-Winkel');
  LblCtl_FacadeTwilightAutomaticEnable                     :FB_BA_Label:=( sObjName:='FRG', sDescr:='Fassaden-Dämmerungsautomatik Freigabe');
  LblCtl_SunProtectionValueOn                              :FB_BA_Label:=( sObjName:='SW_', sDescr:='Sonnenschutz Helligkeitswert Ein');
  LblCtl_SunProtectionValueOff                             :FB_BA_Label:=( sObjName:='SW_', sDescr:='Sonnenschutz Helligkeitswert Aus');
  LblCtl_TimeDelaySunProtectionOn                          :FB_BA_Label:=( sObjName:='ESV', sDescr:='Sonnenschutz Verzögerung Ein');
  LblCtl_TimeDelaySunProtectionOff                         :FB_BA_Label:=( sObjName:='ASV', sDescr:='Sonnenschutz Verzögerung Aus');
  LblCtl_FacadeParkingEnable                               :FB_BA_Label:=( sObjName:='FRG', sDescr:='Fassaden-Parken Freigabe');
  LblCtl_FacadeParkingPosition                             :FB_BA_Label:=( sObjName:='SW_', sDescr:='Fassaden-Parken Position');
  LblCtl_FacadeParkingAngle                                :FB_BA_Label:=( sObjName:='SW_', sDescr:='Fassaden-Parken Winkel');
  LblCtl_WindProtectionState                               :FB_BA_Label:=( sObjName:='STA', sDescr:='Status Sturmschutz');
  LblCtl_SunProtectionState                                :FB_BA_Label:=( sObjName:='STA', sDescr:='Status Sonnenschutz');
//     
  LblCtl_LowWaterMonitor                                   :FB_BA_Label:=( sObjName:='SM_', sDescr:='Wassermangelwächter');
  LblCtl_FireAlert                                         :FB_BA_Label:=( sObjName:='SM_', sDescr:='Feueralarm');
  LblCtl_Burglary                                          :FB_BA_Label:=( sObjName:='SM_', sDescr:='Einbruchalarm');
  LblCtl_CentralSwitchOff                                  :FB_BA_Label:=( sObjName:='ALS', sDescr:='Zentraler Schalter Aus');
  LblCtl_ForcedVentilation                                 :FB_BA_Label:=( sObjName:='ALS', sDescr:='Zwangsbelüftung');
  LblCtl_SmokeExtraction                                   :FB_BA_Label:=( sObjName:='ALS', sDescr:='Entrauchung');
  LblCtl_SetpointIce                                       :FB_BA_Label:=( sObjName:='SW_', sDescr:='Vereisungstemperatur');
  LblCtl_SunProtectionInterval                             :FB_BA_Label:=( sObjName:='SW_', sDescr:='Sonnenschutz Positionierintervall');
  LblCtl_DeiceTime                                         :FB_BA_Label:=( sObjName:='SW_', sDescr:='Vereisungsschutz Enteisungszeit');
  LblCtl_GlobalThermoAutomaticValueOn                      :FB_BA_Label:=( sObjName:='SW_', sDescr:='Thermoautomatik Strahlungswert Ein');
  LblCtl_GlobalThermoAutomaticValueOff                     :FB_BA_Label:=( sObjName:='SW_', sDescr:='Thermoautomatik Strahlungswert Aus');
  LblCtl_GlobalTwilightAutomaticValueOn                    :FB_BA_Label:=( sObjName:='SW_', sDescr:='Dämmerungsautomatik Helligkeitswertwert Ein');
  LblCtl_GlobalTwilightAutomaticValueOff                   :FB_BA_Label:=( sObjName:='SW_', sDescr:='Dämmerungsautomatik Helligkeitswertwert Aus');
  LblCtl_IceAlert                                          :FB_BA_Label:=( sObjName:='SM_', sDescr:='Vereisungsalarm');
  LblCtl_GlobalThermoAutomaticRelease                      :FB_BA_Label:=( sObjName:='FRG', sDescr:='Thermoautomatik Freigabe');
  LblCtl_GlobalTwilightAutomaticRelease                    :FB_BA_Label:=( sObjName:='FRG', sDescr:='Dämmerungsautomatik Freigabe');
  LblCtl_GlobalResetManMode                                :FB_BA_Label:=( sObjName:='ALS', sDescr:='Globaler Reset Handmodus');
  LblCtl_GlobalResetLighting                               :FB_BA_Label:=( sObjName:='ALS', sDescr:='Globaler Reset Lichtfunktionen');
  LblCtl_MaintenanceLighting                               :FB_BA_Label:=( sObjName:='ALS', sDescr:='Wartungschalter Licht');
//     
  LblCtl_BuildingEnergyLevelManual                         :FB_BA_Label:=( sObjName:='BAA', sDescr:='Gebäudeenergieniveau manuelle Auswahl');
  LblCtl_BuildingEnergyLevelActual                         :FB_BA_Label:=( sObjName:='ABA', sDescr:='Gebäudeenergieniveau aktuelle Auswahl');
  LblCtl_BuildingEnergyLevelSched                          :FB_BA_Label:=( sObjName:='ZPL', sDescr:='Gebäudeenergieniveau Zeitschaltplan');
  LblCtl_BuildingModeManual                                :FB_BA_Label:=( sObjName:='BAA', sDescr:='Gebäudebetriebsart manuelle Auswahl');
  LblCtl_BuildingModeActual                                :FB_BA_Label:=( sObjName:='ABA', sDescr:='Gebäudebetriebsart aktuelle Auswahl');
  LblCtl_BuildingModeSched                                 :FB_BA_Label:=( sObjName:='ZPL', sDescr:='Gebäudebetriebsart Zeitschaltplan');
//     
  LblCtl_SummerCompensationX1                              :FB_BA_Label:=( sObjName:='SPX', sDescr:='Sommerkompensation X1');
  LblCtl_SummerCompensationX2                              :FB_BA_Label:=( sObjName:='SPX', sDescr:='Sommerkompensation X2');
  LblCtl_SummerCompensationY1                              :FB_BA_Label:=( sObjName:='SPY', sDescr:='Sommerkompensation Y1');
  LblCtl_SummerCompensationY2                              :FB_BA_Label:=( sObjName:='SPY', sDescr:='Sommerkompensation Y2');
  LblCtl_WinterCompensationX1                              :FB_BA_Label:=( sObjName:='SPX', sDescr:='Winterkompensation X1');
  LblCtl_WinterCompensationX2                              :FB_BA_Label:=( sObjName:='SPX', sDescr:='Winterkompensation X2');
  LblCtl_WinterCompensationY1                              :FB_BA_Label:=( sObjName:='SPY', sDescr:='Winterkompensation Y1');
  LblCtl_WinterCompensationY2                              :FB_BA_Label:=( sObjName:='SPY', sDescr:='Winterkompensation Y2');
  LblCtl_SummerCompensation                                :FB_BA_Label:=( sObjName:='SKP', sDescr:='Sommerkompensation');
  LblCtl_WinterCompensation                                :FB_BA_Label:=( sObjName:='WKP', sDescr:='Winterkompensation');
  LblCtl_SummerCompensationYmin                            :FB_BA_Label:=( sObjName:='SWI', sDescr:='Sommer Kompensation Ymin');
  LblCtl_SummerCompensationYmax                            :FB_BA_Label:=( sObjName:='SWX', sDescr:='Sommer Kompensation Ymax');
  LblCtl_WinterCompensationYmin                            :FB_BA_Label:=( sObjName:='SWI', sDescr:='Winter Kompensation Ymin');
  LblCtl_WinterCompensationYmax                            :FB_BA_Label:=( sObjName:='SWX', sDescr:='Winter Kompensation Ymax');
  LblCtl_SummerCompensationSp                              :FB_BA_Label:=( sObjName:='SWC', sDescr:='Sommer Kompensation Sollwert');
  LblCtl_WinterCompensationSp                              :FB_BA_Label:=( sObjName:='SWC', sDescr:='Winter Kompensation Sollwert');
  LblCtl_SetpointShiftHeating                              :FB_BA_Label:=( sObjName:='SW_', sDescr:='Sollwertverschiebung Heizen');
  LblCtl_SetpointShiftCooling                              :FB_BA_Label:=( sObjName:='SW_', sDescr:='Sollwertverschiebung Kühlen');
  LblCtl_DampConstant                                      :FB_BA_Label:=( sObjName:='SW_', sDescr:='Dämpfungskonstante');
//     
  LblCtl_DelayOn                                           :FB_BA_Label:=( sObjName:='ESV', sDescr:='Einschaltverzögerung');
  LblCtl_DelayOff                                          :FB_BA_Label:=( sObjName:='ASV', sDescr:='Ausschaltverzögerung');
  LblCtl_AntiBlocking                                      :FB_BA_Label:=( sObjName:='BKS', sDescr:='Blockierschutz');
  LblCtl_IdlePeriod                                        :FB_BA_Label:=( sObjName:='ITV', sDescr:='Intervall');
  LblCtl_ImpulsLength                                      :FB_BA_Label:=( sObjName:='IPL', sDescr:='Impulslänge');
  LblCtl_SuppyAirTempSetpointHeaterCalc                    :FB_BA_Label:=( sObjName:='SWC', sDescr:='Zuluft Sw Erhitzer errechnet');
  LblCtl_SuppyAirTempSetpointCoolerCalc                    :FB_BA_Label:=( sObjName:='SWC', sDescr:='Zuluft Sw Kühler errechnet');
  LblCtl_SuppyAirTempSetpointERCCalc                       :FB_BA_Label:=( sObjName:='SWC', sDescr:='Zuluft Sw ERG errechnet');
  LblCtl_X01                                               :FB_BA_Label:=( sObjName:='SWX', sDescr:='Wert Stützpunkt [X1]');
  LblCtl_X02                                               :FB_BA_Label:=( sObjName:='SWX', sDescr:='Wert Stützpunkt [X2]');
  LblCtl_X03                                               :FB_BA_Label:=( sObjName:='SWX', sDescr:='Wert Stützpunkt [X3]');
  LblCtl_X04                                               :FB_BA_Label:=( sObjName:='SWX', sDescr:='Wert Stützpunkt [X4]');
  LblCtl_X05                                               :FB_BA_Label:=( sObjName:='SWX', sDescr:='Wert Stützpunkt [X5]');
  LblCtl_X06                                               :FB_BA_Label:=( sObjName:='SWX', sDescr:='Wert Stützpunkt [X6]');
  LblCtl_X07                                               :FB_BA_Label:=( sObjName:='SWX', sDescr:='Wert Stützpunkt [X7]');
  LblCtl_Y01                                               :FB_BA_Label:=( sObjName:='SWY', sDescr:='Wert Stützpunkt [Y1]');
  LblCtl_Y02                                               :FB_BA_Label:=( sObjName:='SWY', sDescr:='Wert Stützpunkt [Y2]');
  LblCtl_Y02_03                                            :FB_BA_Label:=( sObjName:='SWY', sDescr:='Wert Stützpunkt [Y2-Y3]');
  LblCtl_Y03                                               :FB_BA_Label:=( sObjName:='SWY', sDescr:='Wert Stützpunkt [Y3]');
  LblCtl_Y04                                               :FB_BA_Label:=( sObjName:='SWY', sDescr:='Wert Stützpunkt [Y4]');
  LblCtl_Y05                                               :FB_BA_Label:=( sObjName:='SWY', sDescr:='Wert Stützpunkt [Y5]');
  LblCtl_Y06                                               :FB_BA_Label:=( sObjName:='SWY', sDescr:='Wert Stützpunkt [Y6]');
  LblCtl_Y07                                               :FB_BA_Label:=( sObjName:='SWY', sDescr:='Wert Stützpunkt [Y7]');
  LblCtl_FeedbackMonitoring                                :FB_BA_Label:=( sObjName:='RMW', sDescr:='Rückmeldeüberwachung');
  LblCtl_PreAlarmLimitMAX                                  :FB_BA_Label:=( sObjName:='GWX', sDescr:='Voralarm Grenzwert MAX');
  LblCtl_PreAlarmLimitMIN                                  :FB_BA_Label:=( sObjName:='GWI', sDescr:='Voralarm Grenzwert MIN');
  LblCtl_PreAlarmFault                                     :FB_BA_Label:=( sObjName:='SM_', sDescr:='Voralarm Störung');
  LblCtl_MainAlarmLimitMAX                                 :FB_BA_Label:=( sObjName:='GWX', sDescr:='Hauptalarm Grenzwert MAX');
  LblCtl_MainAlarmLimitMIN                                 :FB_BA_Label:=( sObjName:='GWI', sDescr:='Hauptalarm Grenzwert MIN');
  LblCtl_MainAlarmFault                                    :FB_BA_Label:=( sObjName:='SM_', sDescr:='Hauptalarm Störung');
  LblCtl_ProcPreRinse                                      :FB_BA_LabelProcess:=( sProcessName:='Vorspülen');
  LblCtl_ProjectInfo                                       :FB_BA_Label:=( sObjName:='PI_', sDescr:='Projektinformationen');
//     
  LblCtl_BuildingLighting                                  :FB_BA_Label:=( sObjName:='FEE', sDescr:='Gebäude Lichtsteuerung');
  LblCtl_SetpointLightValue                                :FB_BA_Label:=( sObjName:='SW_', sDescr:='Sollwert Licht');
  LblCtl_SetpointLightTemperature                          :FB_BA_Label:=( sObjName:='SW_', sDescr:='Sollwert Licht-Temperatur');
  LblCtl_SetpointBrightness                                :FB_BA_Label:=( sObjName:='SW_', sDescr:='Sollwert Helligkeit');
  LblCtl_FeedbackLightValue                                :FB_BA_Label:=( sObjName:='RM_', sDescr:='Rückmeldung Licht Stellwert');
  LblCtl_FeedbackLightTemperature                          :FB_BA_Label:=( sObjName:='RM_', sDescr:='Rückmeldung Lichttemperatur');
  LblCtl_FeedbackLightPrio                                 :FB_BA_Label:=( sObjName:='RM_', sDescr:='Rückmeldung Telegrammpriorität');
  LblCtl_ButtonLight                                       :FB_BA_Label:=( sObjName:='TS_', sDescr:='Lichttaster');
//     
  LblCtl_LimitValueWeatherTemperatureSummer                :FB_BA_Label:=( sObjName:='GW_', sDescr:='Grenzwert Witterungstemperatur Sommer');
  LblCtl_LimitValueWeatherTemperatureWinter                :FB_BA_Label:=( sObjName:='GW_', sDescr:='Grenzwert Witterungstemperatur Winter');
  LblCtl_CurrentSequenceTemperature                        :FB_BA_Label:=( sObjName:='STA', sDescr:='Aktuelle Sequenz Temperatur');
  LblCtl_CurrentSequenceHumidity                           :FB_BA_Label:=( sObjName:='STA', sDescr:='Aktuelle Sequenz Feuchte');
END_VAR

// ---- Templates/GVLs/Language/German/LblFunctions_DE.TcGVL
{region '#Template'}
	{attribute 'Version' := '5.0.0.0'}
	{attribute 'Tags' := '"LCID": "1031", "Text": "GVL, AKS, Labels, ObjectName, Description"'}
	{attribute 'Tags' := '"LCID": "1033", "Text": "GVL, DPAD, Labels, ObjectName, Description"'}
	{attribute 'Description' := '"LCID": "1031", "Text": "Anlagenkennzeichnungssystem, Labels functions"'}
	{attribute 'Description' := '"LCID": "1033", "Text": "Data Point Addressing Description, Labels functions"'}
{endregion}

{attribute 'global_init_slot' := '40510'}
VAR_GLOBAL
  LblFun_Requirement                                       :FB_BA_Label:=( sObjName:='AF_', sDescr:='Anforderung');
  LblFun_SystemSwitch                                      :FB_BA_Label:=( sObjName:='ALS', sDescr:='Anlagenschalter');
  LblFun_StatusOccupiedRoom                                :FB_BA_Label:=( sObjName:='BEL', sDescr:='Belegtzustand Raum');
  LblFun_LimitCalculatedValue                              :FB_BA_Label:=( sObjName:='GWC', sDescr:='Berechneter Grenzwert');
  LblFun_SetpointCalculated                                :FB_BA_Label:=( sObjName:='SWC', sDescr:='Berechneter Sollwert');
  LblFun_ReadyForOperation                                 :FB_BA_Label:=( sObjName:='BB_', sDescr:='Betriebsbereit');
  LblFun_OperationalMessage                                :FB_BA_Label:=( sObjName:='BM_', sDescr:='Betriebsmeldung');
  LblFun_HoursOfOperation                                  :FB_BA_Label:=( sObjName:='BZ_', sDescr:='Betriebsstunden');
  LblFun_LimitValueHoursOfOperation                        :FB_BA_Label:=( sObjName:='BZG', sDescr:='Betriebsstunden Grenzwert');
  LblFun_ObjectCalendar                                    :FB_BA_Label:=( sObjName:='CAL', sDescr:='Calendar-Objekt');
  LblFun_ObjectCommand                                     :FB_BA_Label:=( sObjName:='COM', sDescr:='Command-Objekt');
  LblFun_DifferentialConstantController                    :FB_BA_Label:=( sObjName:='TV_', sDescr:='Differenzialkonstante Regler');
  LblFun_SwitchOnErrorUnauthorisedON                       :FB_BA_Label:=( sObjName:='EF_', sDescr:='Einschaltfehler, unerlaubt EIN');
  LblFun_EnergyLevel                                       :FB_BA_Label:=( sObjName:='EN_', sDescr:='Energieniveau');
  LblFun_EnergyLevelCalculated                             :FB_BA_Label:=( sObjName:='ENC', sDescr:='Energieniveau berechnet');
  LblFun_UnlockingDevice                                   :FB_BA_Label:=( sObjName:='ENT', sDescr:='Entriegelung');
  LblFun_ObjectEventEnrollment                             :FB_BA_Label:=( sObjName:='EE_', sDescr:='Event-Enrollment-Objekt');
  LblFun_Enabled                                           :FB_BA_Label:=( sObjName:='FR_', sDescr:='Freigabe');
  LblFun_DangerAlarm                                       :FB_BA_Label:=( sObjName:='GM_', sDescr:='Gefahrmeldung');
  LblFun_Threshold                                         :FB_BA_Label:=( sObjName:='GW_', sDescr:='Grenzwert');
  LblFun_LimitMAX                                          :FB_BA_Label:=( sObjName:='GWX', sDescr:='Grenzwert MAX');
  LblFun_LimitMIN                                          :FB_BA_Label:=( sObjName:='GWI', sDescr:='Grenzwert MIN');
  LblFun_LimitNight                                        :FB_BA_Label:=( sObjName:='GWN', sDescr:='Grenzwert Nacht');
  LblFun_LimitDay                                          :FB_BA_Label:=( sObjName:='GWT', sDescr:='Grenzwert Tag');
  LblFun_ObjectGroup                                       :FB_BA_Label:=( sObjName:='GP_', sDescr:='Group-Objekt');
  LblFun_localPriorityAndOperatingUnitsManualMessage       :FB_BA_Label:=( sObjName:='HD_', sDescr:='LVB-Handmeldung');
  LblFun_HeatingCharacteristicCurveExponent                :FB_BA_Label:=( sObjName:='HEX', sDescr:='Heizkennlinie Exponent');
  LblFun_HeatingCharacteristicCurveParallelDisplacement    :FB_BA_Label:=( sObjName:='HPV', sDescr:='Heizkennlinie Parallelverschiebung');
  LblFun_HeatingCharacteristicCurveSteepness               :FB_BA_Label:=( sObjName:='HST', sDescr:='Heizkennlinie Steilheit');
  LblFun_HeatingCircuitNightReduction                      :FB_BA_Label:=( sObjName:='NAH', sDescr:='Heizkreis Nachtabsenkung');
  LblFun_Hysteresis                                        :FB_BA_Label:=( sObjName:='HYS', sDescr:='Hysterese');
  LblFun_Calendar                                          :FB_BA_Label:=( sObjName:='KAL', sDescr:='Kalender');
  LblFun_RuntimeError                                      :FB_BA_Label:=( sObjName:='LFZ', sDescr:='Laufzeitfehler');
  LblFun_LoopMAXLimit                                      :FB_BA_Label:=( sObjName:='LPX', sDescr:='Loop-MAX-Begrenzung');
  LblFun_LoopMINLimit                                      :FB_BA_Label:=( sObjName:='LPI', sDescr:='Loop-MIN-Begrenzung');
  LblFun_LoopObject                                        :FB_BA_Label:=( sObjName:='LP_', sDescr:='Regler');
  LblFun_LoopObjectCascadeSupplyAirTemperature             :FB_BA_Label:=( sObjName:='LP_', sDescr:='Führungsregler Zulufttemperatur');
  LblFun_LoopObjectCascadeSupplyAirHumidity                :FB_BA_Label:=( sObjName:='LP_', sDescr:='Führungsregler Zuluftfeuchte');
  LblFun_MaximumValue                                      :FB_BA_Label:=( sObjName:='MAX', sDescr:='Maximalwert');
  LblFun_MeasuredValue                                     :FB_BA_Label:=( sObjName:='MW_', sDescr:='Messwert');
  LblFun_MeasuredValueCalculated                           :FB_BA_Label:=( sObjName:='MWC', sDescr:='Berechneter Messwert');
  LblFun_MeasuredValueEast                                 :FB_BA_Label:=( sObjName:='MW_', sDescr:='Messwert Osten');
  LblFun_MeasuredValueNorth                                :FB_BA_Label:=( sObjName:='MW_', sDescr:='Messwert Norden');
  LblFun_MeasuredValueSouth                                :FB_BA_Label:=( sObjName:='MW_', sDescr:='Messwert Sueden');
  LblFun_MeasuredValueWest                                 :FB_BA_Label:=( sObjName:='MW_', sDescr:='Messwert Westen');
  LblFun_MinimumValue                                      :FB_BA_Label:=( sObjName:='MIN', sDescr:='Minimalwert');
  LblFun_Mean                                              :FB_BA_Label:=( sObjName:='MWT', sDescr:='Mittelwert');
  LblFun_FollowUpTime                                      :FB_BA_Label:=( sObjName:='NL_', sDescr:='Nachlaufzeit');
  LblFun_ResetTime                                         :FB_BA_Label:=( sObjName:='TN_', sDescr:='Nachstellzeit');
  LblFun_FeedbackDelay                                     :FB_BA_Label:=( sObjName:='ZVR', sDescr:='Zeitverzögerung Rückmeldung');
  LblFun_ObjectNotificationClass                           :FB_BA_Label:=( sObjName:='NC_', sDescr:='Notification-Class-Objekt');
  LblFun_EventClassObject                                  :FB_BA_Label:=( sObjName:='EKL', sDescr:='Ereignisklasse');
  LblFun_Programobject                                     :FB_BA_Label:=( sObjName:='PRG', sDescr:='Programm');
  LblFun_ProportionalBand                                  :FB_BA_Label:=( sObjName:='XP_', sDescr:='Proportionalband');
  LblFun_FeedbackOPEN                                      :FB_BA_Label:=( sObjName:='RMA', sDescr:='Rückmeldung AUF');
  LblFun_FeedbackCLOSED                                    :FB_BA_Label:=( sObjName:='RMZ', sDescr:='Rückmeldung ZU');
  LblFun_FeedbackValue                                     :FB_BA_Label:=( sObjName:='RW_', sDescr:='Rückführwert');
  LblFun_FeedbackErrorOPEN                                 :FB_BA_Label:=( sObjName:='RFA', sDescr:='Rückmeldefehler AUF');
  LblFun_FeedbackErrorCLOSED                               :FB_BA_Label:=( sObjName:='RFZ', sDescr:='Rückmeldefehler ZU');
  LblFun_Feedback                                          :FB_BA_Label:=( sObjName:='RM_', sDescr:='Rückmeldung');
  LblFun_ExecutionControl                                  :FB_BA_Label:=( sObjName:='RF_', sDescr:='Ausführkontrolle');
  LblFun_SwitchingCommand                                  :FB_BA_Label:=( sObjName:='SB_', sDescr:='Schaltbefehl');
  LblFun_Scheduler                                         :FB_BA_Label:=( sObjName:='ZPL', sDescr:='Zeitschaltplan');
  LblFun_Setpoint                                          :FB_BA_Label:=( sObjName:='SW_', sDescr:='Sollwert');
  LblFun_SetpointComfortHeating                            :FB_BA_Label:=( sObjName:='SW_', sDescr:='Sollwert Comfort Heizen');
  LblFun_SetpointPreComfortHeating                         :FB_BA_Label:=( sObjName:='SW_', sDescr:='Sollwert Pre-comfort Heizen');
  LblFun_SetpointEconomyHeating                            :FB_BA_Label:=( sObjName:='SW_', sDescr:='Sollwert Economy Heizen');
  LblFun_SetpointProtectionHeating                         :FB_BA_Label:=( sObjName:='SW_', sDescr:='Sollwert Protection Heizen');
  LblFun_SetpointComfortCooling                            :FB_BA_Label:=( sObjName:='SW_', sDescr:='Sollwert Comfort Kühlen');
  LblFun_SetpointPreComfortCooling                         :FB_BA_Label:=( sObjName:='SW_', sDescr:='Sollwert Pre-comfort Kühlen');
  LblFun_SetpointEconomyCooling                            :FB_BA_Label:=( sObjName:='SW_', sDescr:='Sollwert Economy Kühlen');
  LblFun_SetpointProtectionCooling                         :FB_BA_Label:=( sObjName:='SW_', sDescr:='Sollwert Protection Kühlen');
  LblFun_SetpointBase                                      :FB_BA_Label:=( sObjName:='SWB', sDescr:='Basissollwert');
  LblFun_SetpointHeating                                   :FB_BA_Label:=( sObjName:='SWH', sDescr:='Sollwert Heizen');
  LblFun_SetpointCooling                                   :FB_BA_Label:=( sObjName:='SWK', sDescr:='Sollwert Kühlen');
  LblFun_SetpointMaximum                                   :FB_BA_Label:=( sObjName:='SWX', sDescr:='Sollwert, maximal');
  LblFun_SetpointMechanical                                :FB_BA_Label:=( sObjName:='SWM', sDescr:='Sollwert, mechanisch');
  LblFun_SetpointMinimum                                   :FB_BA_Label:=( sObjName:='SWI', sDescr:='Sollwert, minimal');
  LblFun_SetpointNight                                     :FB_BA_Label:=( sObjName:='SWN', sDescr:='Sollwert Nacht');
  LblFun_SetpointDay                                       :FB_BA_Label:=( sObjName:='SWT', sDescr:='Sollwert Tag');
  LblFun_SetpointAdjuster                                  :FB_BA_Label:=( sObjName:='SWV', sDescr:='Sollwertversteller');
  LblFun_SetpointAdjustmentMechanical                      :FB_BA_Label:=( sObjName:='SVM', sDescr:='Sollwertverstellung, mechanisch');
  LblFun_Selection                                         :FB_BA_Label:=( sObjName:='AUS', sDescr:='Auswahl');
  LblFun_Status                                            :FB_BA_Label:=( sObjName:='STA', sDescr:='Status');
  LblFun_ControlSignal                                     :FB_BA_Label:=( sObjName:='ST_', sDescr:='Stellsignal');
  LblFun_Fault                                             :FB_BA_Label:=( sObjName:='SM_', sDescr:='Störung');
  LblFun_FaultFuse                                         :FB_BA_Label:=( sObjName:='SM_', sDescr:='Sicherung Störung ');
  LblFun_Button                                            :FB_BA_Label:=( sObjName:='TS_', sDescr:='Taster');
  LblFun_DeadZone                                          :FB_BA_Label:=( sObjName:='TZ_', sDescr:='Totzone');
  LblFun_ObjectTrendLogMultiple                            :FB_BA_Label:=( sObjName:='TRM', sDescr:='Trend-Log-Multiple-Objekt');
  LblFun_ObjectTrendLog                                    :FB_BA_Label:=( sObjName:='TR_', sDescr:='Trend-Log-Objekt');
  LblFun_AmplificationController                           :FB_BA_Label:=( sObjName:='KP_', sDescr:='Verstärkung Regler');
  LblFun_RetentionPeriod                                   :FB_BA_Label:=( sObjName:='TV_', sDescr:='Vorhaltezeit');
  LblFun_MaintenanceMessage                                :FB_BA_Label:=( sObjName:='WM_', sDescr:='Wartungsmeldung');
  LblFun_Efficiency                                        :FB_BA_Label:=( sObjName:='WG_', sDescr:='Wirkungsgrad');
  LblFun_CountValue                                        :FB_BA_Label:=( sObjName:='ZW_', sDescr:='Zählwert');
  LblFun_TimeProgram                                       :FB_BA_Label:=( sObjName:='ZPR', sDescr:='Zeitprogramm');
//     Beckhoff Skalierung
  LblFun_ValueX1                                           :FB_BA_Label:=( sObjName:='SPX', sDescr:='Wert Stützpunkt [X1]');
  LblFun_ValueX2                                           :FB_BA_Label:=( sObjName:='SPX', sDescr:='Wert Stützpunkt [X2]');
  LblFun_ValueX3                                           :FB_BA_Label:=( sObjName:='SPX', sDescr:='Wert Stützpunkt [X3]');
  LblFun_ValueX4                                           :FB_BA_Label:=( sObjName:='SPX', sDescr:='Wert Stützpunkt [X4]');
  LblFun_ValueX5                                           :FB_BA_Label:=( sObjName:='SPX', sDescr:='Wert Stützpunkt [X5]');
  LblFun_ValueX6                                           :FB_BA_Label:=( sObjName:='SPX', sDescr:='Wert Stützpunkt [X6]');
  LblFun_ValueX7                                           :FB_BA_Label:=( sObjName:='SPX', sDescr:='Wert Stützpunkt [X7]');
  LblFun_ValueY1                                           :FB_BA_Label:=( sObjName:='SPY', sDescr:='Wert Stützpunkt [Y1]');
  LblFun_ValueY2                                           :FB_BA_Label:=( sObjName:='SPY', sDescr:='Wert Stützpunkt [Y2]');
  LblFun_ValueY3                                           :FB_BA_Label:=( sObjName:='SPY', sDescr:='Wert Stützpunkt [Y3]');
  LblFun_ValueY2_3                                         :FB_BA_Label:=( sObjName:='SPY', sDescr:='Wert Stützpunkt [Y2-Y3]');
  LblFun_ValueY4                                           :FB_BA_Label:=( sObjName:='SPY', sDescr:='Wert Stützpunkt [Y4]');
  LblFun_ValueY5                                           :FB_BA_Label:=( sObjName:='SPY', sDescr:='Wert Stützpunkt [Y5]');
  LblFun_ValueY6                                           :FB_BA_Label:=( sObjName:='SPY', sDescr:='Wert Stützpunkt [Y6]');
  LblFun_ValueY7                                           :FB_BA_Label:=( sObjName:='SPY', sDescr:='Wert Stützpunkt [Y7]');
  LblFun_SuppyAirTempSetpointHeaterCalc                    :FB_BA_Label:=( sObjName:='SWC', sDescr:='Zulufttemperatursollwert Erhitzer errechnet');
  LblFun_SuppyAirTempSetpointCoolerCalc                    :FB_BA_Label:=( sObjName:='SWC', sDescr:='Zulufttemperatursollwert Kühler errechnet');
  LblFun_SuppyAirTempSetpointERCCalc                       :FB_BA_Label:=( sObjName:='SWC', sDescr:='Zulufttemperatursollwert ERG errechnet');
//     Beckhoff Raumautomation
  LblFun_FireAlert                                         :FB_BA_Label:=( sObjName:='GM_', sDescr:='Feueralarm');
  LblFun_Burglary                                          :FB_BA_Label:=( sObjName:='GM_', sDescr:='Einbruchalarm');
  LblFun_CentralSwitchOff                                  :FB_BA_Label:=( sObjName:='ALS', sDescr:='Zentraler Schalter Aus');
  LblFun_LightAreaModeManual                               :FB_BA_Label:=( sObjName:='BAA', sDescr:='Bereichsbetriebsart manuelle Auswahl');
  LblFun_LightAreaModeActual                               :FB_BA_Label:=( sObjName:='ABA', sDescr:='Bereichsbetriebsart aktuelle Auswahl');
  LblFun_LightAreaModeSched                                :FB_BA_Label:=( sObjName:='ZPL', sDescr:='Bereichsbetriebsart Zeitschaltplan');
  LblFun_SunPrtcPosition                                   :FB_BA_Label:=( sObjName:='RM_', sDescr:='Sonnenschutz errechnete Position');
  LblFun_SunPrtcAngle                                      :FB_BA_Label:=( sObjName:='RM_', sDescr:='Sonnenschutz errechneter Winkel');
  LblFun_FeedbackLightValue                                :FB_BA_Label:=( sObjName:='RM_', sDescr:='Rückmeldung Licht Stellwert');
  LblFun_FeedbackSunblindPosition                          :FB_BA_Label:=( sObjName:='RM_', sDescr:='Rückmeldung Sonnenschutz Position');
  LblFun_FeedbackSunblindAngle                             :FB_BA_Label:=( sObjName:='RM_', sDescr:='Rückmeldung Sonnenschutz Winkel');
END_VAR

// ---- Templates/GVLs/Language/German/LblPlant_DE.TcGVL
{region '#Template'}
	{attribute 'Version' := '5.0.1.0'}
	{attribute 'Tags' := '"LCID": "1031", "Text": "GVL, DPAD, Plants, ObjectName, Description"'}
	{attribute 'Tags' := '"LCID": "1033", "Text": "GVL, DPAD, Plants, ObjectName, Description"'}
	{attribute 'Description' := '"LCID": "1031", "Text": "Textliste Anlagen"'}
	{attribute 'Description' := '"LCID": "1033", "Text": "Text list plants"'}
{endregion}


